(* CODESYS project Warehouse.project

Project tree, tasks and I/O mapping:
  PLC_AC500_V2 : AC500 PM554-ETH, ABB Automation Products GmbH, order no. 1SAP120600R0071, version 2.8.0.0
      settings: PM5xx Type = PM554-ETH; CoDeSys V2.3 Target = 23844; Product version = [2, 2, 0, 5]
    Application
      application App
        global variables GVL
        Library_Manager
    OBIO : 8DI+6DO, ABB Automation Products GmbH, version 2.8.0.0
        unmapped channels: Digital inputs DI0 - DI7, Interrupt DI0 - DI3, State Byte PWM 2, State Byte PWM 3, Unused, Unused, Unused, Unused, Unused, Unused, Unused, Unused, Unused, Unused, Unused, Unused, Unused, Unused, Unused, Actual value 1, Actual value 2, State Byte 1, State Byte 2, Digital outputs DO0 / NO0 - DO5 / NO5, Control Byte PWM 2, PWM 2, frequency / cycle time, PWM 2, duty cycle / duty time, Control Byte PWM 3, Unused, PWM 3, frequency / cycle time, PWM 3, duty cycle / duty time, Unused, Unused, Unused, Unused, Unused, Unused, Unused, Unused, Unused,
          Unused, Unused, Unused, Start value 1, End value 1, Start value 2, End value 2, Control Byte 1, Control Byte 2
    IO_Bus : I/O-Bus, ABB Automation Products GmbH, version 2.8.0.0
      DC532 : DC532, ABB Automation Products GmbH, order no. 1SAPx40100R0001, version 2.8.0.0
          input  XposRight : BOOL  // Digital inputs I0 - I15.Bytes.Digital inputs I0 - I7.Digital input I0
          input  XposMid : BOOL  // Digital inputs I0 - I15.Bytes.Digital inputs I0 - I7.Digital input I1
          input  XposLeft : BOOL  // Digital inputs I0 - I15.Bytes.Digital inputs I0 - I7.Digital input I2
          input  YposIn : BOOL  // Digital inputs I0 - I15.Bytes.Digital inputs I0 - I7.Digital input I3
          input  YposMid : BOOL  // Digital inputs I0 - I15.Bytes.Digital inputs I0 - I7.Digital input I4
          input  YposOut : BOOL  // Digital inputs I0 - I15.Bytes.Digital inputs I0 - I7.Digital input I5
          input  Zpos3above : BOOL  // Digital inputs I0 - I15.Bytes.Digital inputs I0 - I7.Digital input I6
          input  Zpos3below : BOOL  // Digital inputs I0 - I15.Bytes.Digital inputs I0 - I7.Digital input I7
          input  Zpos2above : BOOL  // Digital inputs I0 - I15.Bytes.Digital inputs I8 - I15.Digital input I8
          input  Zpos2below : BOOL  // Digital inputs I0 - I15.Bytes.Digital inputs I8 - I15.Digital input I9
          input  Zpos1above : BOOL  // Digital inputs I0 - I15.Bytes.Digital inputs I8 - I15.Digital input I10
          input  Zpos1below : BOOL  // Digital inputs I0 - I15.Bytes.Digital inputs I8 - I15.Digital input I11
          input  FeederOccupied : BOOL  // Digital inputs I0 - I15.Bytes.Digital inputs I8 - I15.Digital input I12
          input  HandKey1 : BOOL  // Digital inputs I0 - I15.Bytes.Digital inputs I8 - I15.Digital input I13
          input  HandKey2 : BOOL  // Digital inputs I0 - I15.Bytes.Digital inputs I8 - I15.Digital input I14
          output XRight : BOOL  // Digital outputs C16 - C31.Bytes.Digital outputs C24 - C31.Digital output C24
          output XLeft : BOOL  // Digital outputs C16 - C31.Bytes.Digital outputs C24 - C31.Digital output C25
          output Yin : BOOL  // Digital outputs C16 - C31.Bytes.Digital outputs C24 - C31.Digital output C26
          output Yout : BOOL  // Digital outputs C16 - C31.Bytes.Digital outputs C24 - C31.Digital output C27
          output Zup : BOOL  // Digital outputs C16 - C31.Bytes.Digital outputs C24 - C31.Digital output C28
          output Zdown : BOOL  // Digital outputs C16 - C31.Bytes.Digital outputs C24 - C31.Digital output C29
          output Led1 : BOOL  // Digital outputs C16 - C31.Bytes.Digital outputs C24 - C31.Digital output C30
          output Led2 : BOOL  // Digital outputs C16 - C31.Bytes.Digital outputs C24 - C31.Digital output C31
          unmapped channels: Digital inputs I0 - I15, Digital inputs C16 - C31, Digital outputs C16 - C31, Actual value 1, Actual value 2, State Byte 1, State Byte 2, Start value 1, End value 1, Start value 2, End value 2, Control Byte 1, Control Byte 2, Digital inputs I0 - I15, Digital inputs C16 - C31, Digital outputs C16 - C31, Digital inputs I0 - I15, Digital inputs C16 - C31, Digital outputs C16 - C31
    Interfaces : Interfaces, ABB Automation Products GmbH, version 2.8.0.0
      COM1_Online_Access : COM1 - Online Access, ABB Automation Products GmbH, version 2.8.0.0
      COM2_None : COM2 - None, ABB Automation Products GmbH, version 2.8.0.0
      Ethernet : Onboard Ethernet, ABB Automation Products GmbH, version 2.8.0.0
        ETH1 : ETH1, ABB Automation Products GmbH, version 2.8.0.0
        Protocols : Protocols, ABB Automation Products GmbH, version 2.8.0.0
          Modbus_TCP_IP_Server : Modbus TCP/IP Server, ABB Automation Products GmbH, version 2.8.0.0
  visualisation Visualization
  text list GlobalTextList
  visualisation Visualization_1
  program PLC_PRG [ST]
*)

// PLC_AC500_V2/Application/App/GVL
{attribute 'qualified_only'}
VAR_GLOBAL
	reset: BOOL:= FALSE;
	reset_UI: BOOL:= FALSE;
	reset_UnLoading: BOOL:= FALSE;
	reset_Loading: BOOL:= FALSE;
	Count_Enable: BOOL:= FALSE;
	Reset_Count: BOOL:=TRUE;
	Count_X:INT:=0;
	Count_Z:INT:=0;	
	Tap_X:BOOL:=FALSE;
	Tap_Z:BOOL:=FALSE;
	State_X_1: BOOL:=FALSE;
	State_X_2: BOOL:=FALSE;
	State_X_3: BOOL:=FALSE;
	State_Z_1: BOOL:=FALSE;
	State_Z_2: BOOL:=FALSE;
	State_Z_3: BOOL:=FALSE;
	reset_home: BOOL:=FALSE;
	CountX_4: BOOL:=FALSE;
	CountZ_4: BOOL:=FALSE;
	Loading: BOOL:=FALSE;
	State_1_1: BOOL:=FALSE;
	State_1_2: BOOL:=FALSE;
	State_1_3: BOOL:=FALSE;
	State_2_1: BOOL:=FALSE;
	State_2_2: BOOL:=FALSE;
	State_2_3: BOOL:=FALSE;
	State_3_1: BOOL:=FALSE;
	State_3_2: BOOL:=FALSE;
	State_3_3: BOOL:=FALSE;
	HMI: BOOL:=FALSE;
	Manual: BOOL:=FALSE;
END_VAR

// PLC_PRG
PROGRAM PLC_PRG
VAR
	STATE:INT:=0;
	endInit:BOOL:=FALSE;
END_VAR

CASE State OF
	0:
		Init(endInit1 =>  endInit);
		IF endInit THEN
			endInit:= FALSE;
			reset_Loading:= TRUE;
			reset_UnLoading:=TRUE;
			STATE := 1;
		END_IF

	1:
		UI(UI_END =>  endInit);
		IF endInit THEN
			endInit:= FALSE;
			STATE := 2;
			Count_X:=0;
			Count_Z:=0;
		END_IF

	2:
		IF State_X_1 AND State_Z_1 THEN
			Loading11(step6 =>  endInit);
		ELSIF State_X_1 AND State_Z_2 THEN
			Loading12(step6 =>  endInit);
		ELSIF State_X_1 AND State_Z_3 THEN
			Loading13(step6 =>  endInit);
		ELSIF State_X_2 AND State_Z_1 THEN
			Loading21(step6 =>  endInit);
		ELSIF State_X_2 AND State_Z_2 THEN
			Loading22(step6 =>  endInit);
		ELSIF State_X_2 AND State_Z_3 THEN
			Loading23(step6 =>  endInit);
		ELSIF State_X_3 AND State_Z_1 THEN
			Loading31(step6 =>  endInit);
		ELSIF State_X_3 AND State_Z_2 THEN
			Loading32(step6 =>  endInit);
		ELSIF State_X_3 AND State_Z_3 THEN
			Loading33(step6 =>  endInit);
		END_IF

		IF endInit THEN
			endInit:= FALSE;
			STATE := 3;
			reset:=TRUE;
			reset_UI:=TRUE;
			reset_home:=TRUE;
		END_IF

	3:
		initHome(endInit1 =>  endInit);
		IF endInit THEN
			reset_Loading:= TRUE;
			reset_UnLoading:=TRUE;
			endInit:= FALSE;

			STATE := 4;
		END_IF

	4:
		UI(UI_END =>  endInit);
		IF endInit THEN
			endInit:= FALSE;
			STATE := 5;
			Count_X:=0;
			Count_Z:=0;
		END_IF

	5:
		IF State_X_1 AND State_Z_1 THEN
			Unloading11(step6 =>  endInit);
		ELSIF State_X_1 AND State_Z_2 THEN
			Unloading12(step6 =>  endInit);
		ELSIF State_X_1 AND State_Z_3 THEN
			Unloading13(step6 =>  endInit);
		ELSIF State_X_2 AND State_Z_1 THEN
			Unloading21(step7 =>  endInit);
		ELSIF State_X_2 AND State_Z_2 THEN
			Unloading22(step7 =>  endInit);
		ELSIF State_X_2 AND State_Z_3 THEN
			Unloading23(step7 =>  endInit);
		ELSIF State_X_3 AND State_Z_1 THEN
			Unloading31(step7 =>  endInit);
		ELSIF State_X_3 AND State_Z_2 THEN
			Unloading32(step7 =>  endInit);
		ELSIF State_X_3 AND State_Z_3 THEN
			Unloading33(step7 =>  endInit);
		END_IF

		IF endInit THEN
			endInit:= FALSE;
			STATE := 6;
			reset:=TRUE;
			reset_UI:=TRUE;
			reset_home:=TRUE;
		END_IF

	6:
		initHome(endInit1 =>  endInit);
		IF endInit THEN
			reset_Loading:= TRUE;
			reset_UnLoading:=TRUE;
			endInit:= FALSE;
			STATE := 1;
		END_IF

END_CASE

END_PROGRAM

// /Visualization
VISUALIZATION Visualization  // 2x2
END_VISUALIZATION

// /Visualization_1
VISUALIZATION Visualization_1  // 2x2
END_VISUALIZATION
